// SIMATIC S7-200 project (STEP 7-Micro/WIN), CPU 221 REL 01.10

SYMBOL_TABLE USER1
S0               I0.0     // cong tac khoi dong he thong lam viec
S1               I0.1     // nut khoi dong dong co
S2               I0.2     // nut dung he thong
F3               I0.3     // do le nhiet bao ve he thong
M1               Q0.0     // dong co M1
H0               Q0.1     // den bao he thong lam viec
END_SYMBOL_TABLE

ORGANIZATION_BLOCK MAIN:OB1
TITLE=PROGRAM COMMENTS
BEGIN
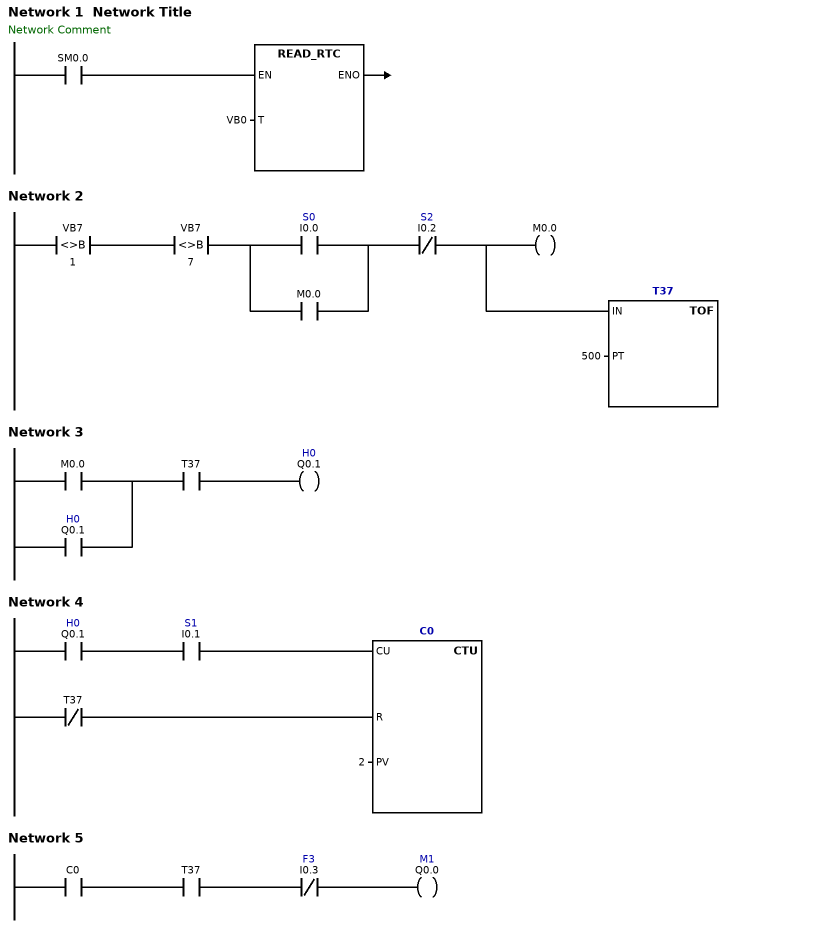
Network 1 // Network Title
// Network Comment
LD     SM0.0
TODR   VB0
Network 2
LDB<>  VB7, 1
AB<>   VB7, 7
LD     S0:I0.0
O      M0.0
ALD
AN     S2:I0.2
=      M0.0
TOF    T37, 500
Network 3
LD     M0.0
O      H0:Q0.1
A      T37
=      H0:Q0.1
Network 4
LD     H0:Q0.1
A      S1:I0.1
LDN    T37
CTU    C0, 2
Network 5
LD     C0
A      T37
AN     F3:I0.3
=      M1:Q0.0
END_ORGANIZATION_BLOCK
